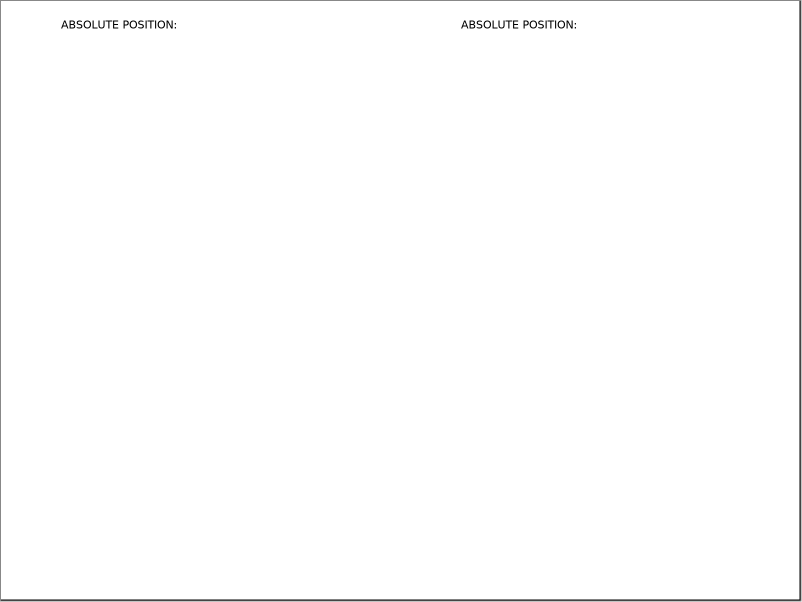
VISUALIZATION F23_Cam_Table_Select  // 802x602
    Rectangle (0,0 800x600)
    Label (10,10 170x30), "ABSOLUTE POSITION:"
    Label (410,10 170x30), "ABSOLUTE POSITION:"
END_VISUALIZATION

(* stored: Version 1.1.0.1, ProductVersion 3.1.4022.7
   Visu F23_Cam_Table_Select: Id {f72eb608-a5b3-4b13-90d6-768c74aa40d5} *)
